// TIA Portal V20 export
TYPE "LER_SignalsInput"
// stored: Access Published
   STRUCT
      "Button Left" : Array[0..15] of Bool;
      "Button Right" : Array[0..15] of Bool;
   END_STRUCT;
END_TYPE
